PROGRAM prg_DynamischVerschalen
VAR
	nPotentioMeter		AT		%I*		:INT;
	
	nPotPower			AT		%Q*		:INT := 32767; //Potentiometer voeden met 5V
	nWaarde				AT		%Q*		:REAL;
	nScaledMax			AT		%Q*		:INT;
END_VAR

nScaledMax := 10;
nWaarde := INT_TO_REAL(nPotentioMeter) * INT_TO_REAL(nScaledMax) / 32767;

//Andere oplossing:
//nScaledMax := 10;
//nWaarde := INT_TO_REAL(nPotentioMeter) * nScaledMax) / 32767;

END_PROGRAM

(* stored: Version 1.1.0.1, ProductVersion 3.1.4024.15
   POU prg_DynamischVerschalen: Id {010acd25-5d1e-456e-9bef-2c5ae678a5bc}, SpecialFunc None *)
